TYPE ST_mcAxisNC :
STRUCT
	lrActPosition			:		LREAL;
	lrActVelocity			:		LREAL;
	lrActTorque				:		LREAL;
	lrMotorTemp				:		LREAL;
END_STRUCT
END_TYPE

(* stored: Version 1.1.0.1, ProductVersion 3.1.4024.6
   DUT ST_mcAxisNC: Id {d82da8bd-d902-4711-9062-8c2fe10cabf8} *)
